FUNCTION_BLOCK L4_FMS205_F3SeqFin_SFC EXTENDS L1_ControllerBase_SFC
// Girar 8 veces el plato para determinar qué tipo de tapa hay en cada sector del plato
VAR_INPUT
	TapasOk			: BOOL;
END_VAR

VAR_IN_OUT
	Evacu		 	: L3_Evacuador;
	Plato			: L3_PlatoDivisor;
END_VAR

VAR_OUTPUT
	InitTapas		: BOOL;
	Giros 			: INT := 0;
END_VAR

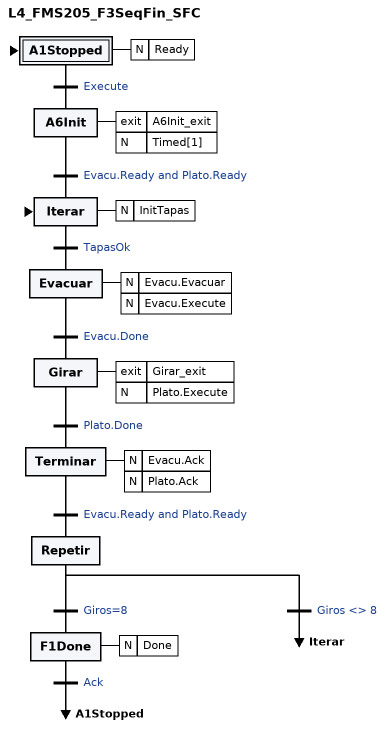
INITIAL_STEP A1Stopped:
    Ready(N);
END_STEP
TRANSITION FROM A1Stopped TO A6Init
    := Execute;
END_TRANSITION
STEP A6Init:
    A6Init_exit(P0);  // exit action
    Timed[1](N);
END_STEP
TRANSITION FROM A6Init TO Iterar
    := Evacu.Ready and Plato.Ready;
END_TRANSITION
STEP Iterar:
    InitTapas(N);
END_STEP
TRANSITION FROM Iterar TO Evacuar
    := TapasOk;
END_TRANSITION
STEP Evacuar:
    Evacu.Evacuar(N);
    Evacu.Execute(N);
END_STEP
TRANSITION FROM Evacuar TO Girar
    := Evacu.Done;
END_TRANSITION
STEP Girar:
    Girar_exit(P0);  // exit action
    Plato.Execute(N);
END_STEP
TRANSITION FROM Girar TO Terminar
    := Plato.Done;
END_TRANSITION
STEP Terminar:
    Evacu.Ack(N);
    Plato.Ack(N);
END_STEP
TRANSITION FROM Terminar TO Repetir
    := Evacu.Ready and Plato.Ready;
END_TRANSITION
STEP Repetir:
END_STEP
TRANSITION FROM Repetir TO F1Done
    := Giros=8;
END_TRANSITION
TRANSITION FROM Repetir TO Iterar
    := Giros <> 8;
END_TRANSITION
STEP F1Done:
    Done(N);
END_STEP
TRANSITION FROM F1Done TO A1Stopped
    := Ack;
END_TRANSITION

ACTION A6Init_exit:
Giros:=0;
END_ACTION

ACTION Girar_exit:
Giros:=Giros+1;
END_ACTION

END_FUNCTION_BLOCK

(* stored: Version 1.1.0.1, ProductVersion 3.1.4024.11
   POU L4_FMS205_F3SeqFin_SFC: Id {22407fab-8c54-4f66-ad2d-4fd58091b013}, SpecialFunc None
   Action A6Init_exit: Id {266d0edc-df9f-4d5a-b150-0890e400ec7f}
   Action Girar_exit: Id {2f34e197-f97c-49e5-b0de-c3efbfb39099} *)
